// TIA Portal V19 export
TYPE "LEXCHANGETRAY_typeConstraintWorkstationEm_toConstraintRollerReq"
// stored: Access Published
   STRUCT
      transferEnable : Bool;   // 请求转移
   END_STRUCT;
END_TYPE
